FUNCTION_BLOCK GUYSON_PRG_SEL
VAR_INPUT

	US_ON_BOOL		:BOOL; 		(*ULTRASONIC ON/OFF BIT*)
	PRG_ADD_INT		:INT;		(*PROGRAM ADDRESS*)


END_VAR
VAR_OUTPUT

	BOOL_US_BIT1		:BOOL; 		(*ULTRASONIC EXT1*)
	BOOL_US_BIT2		:BOOL; 		(*ULTRASONIC EXT2*)
	BOOL_US_BIT3		:BOOL; 		(*ULTRASONIC EXT3*)


END_VAR
VAR
END_VAR

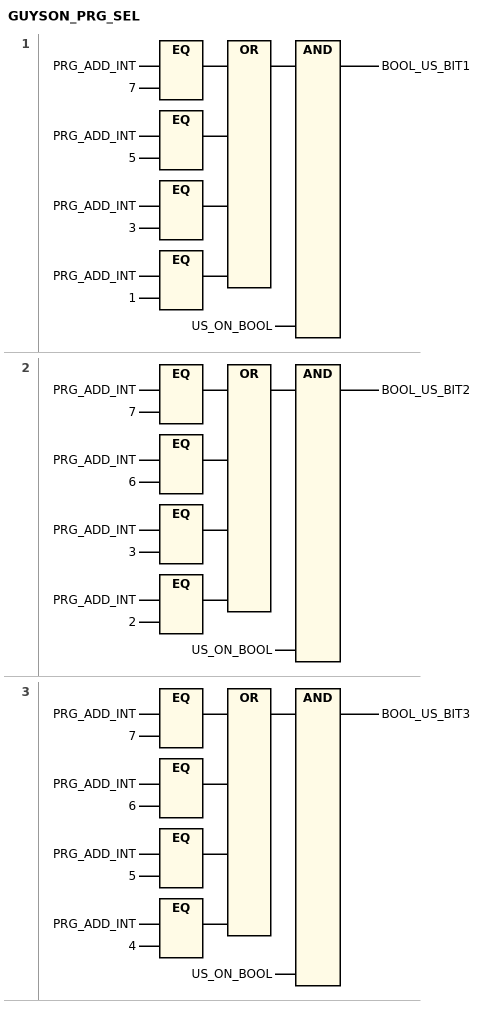
// NETWORK 1
BOOL_US_BIT1 := (PRG_ADD_INT = 7 OR PRG_ADD_INT = 5 OR PRG_ADD_INT = 3 OR PRG_ADD_INT = 1) AND US_ON_BOOL;

// NETWORK 2
BOOL_US_BIT2 := (PRG_ADD_INT = 7 OR PRG_ADD_INT = 6 OR PRG_ADD_INT = 3 OR PRG_ADD_INT = 2) AND US_ON_BOOL;

// NETWORK 3
BOOL_US_BIT3 := (PRG_ADD_INT = 7 OR PRG_ADD_INT = 6 OR PRG_ADD_INT = 5 OR PRG_ADD_INT = 4) AND US_ON_BOOL;

END_FUNCTION_BLOCK

(* stored: Version 1.1.0.1, ProductVersion 3.1.4024.12
   POU GUYSON_PRG_SEL: Id {01048b71-a775-4830-9b9d-1210eb88b934}, SpecialFunc None *)
